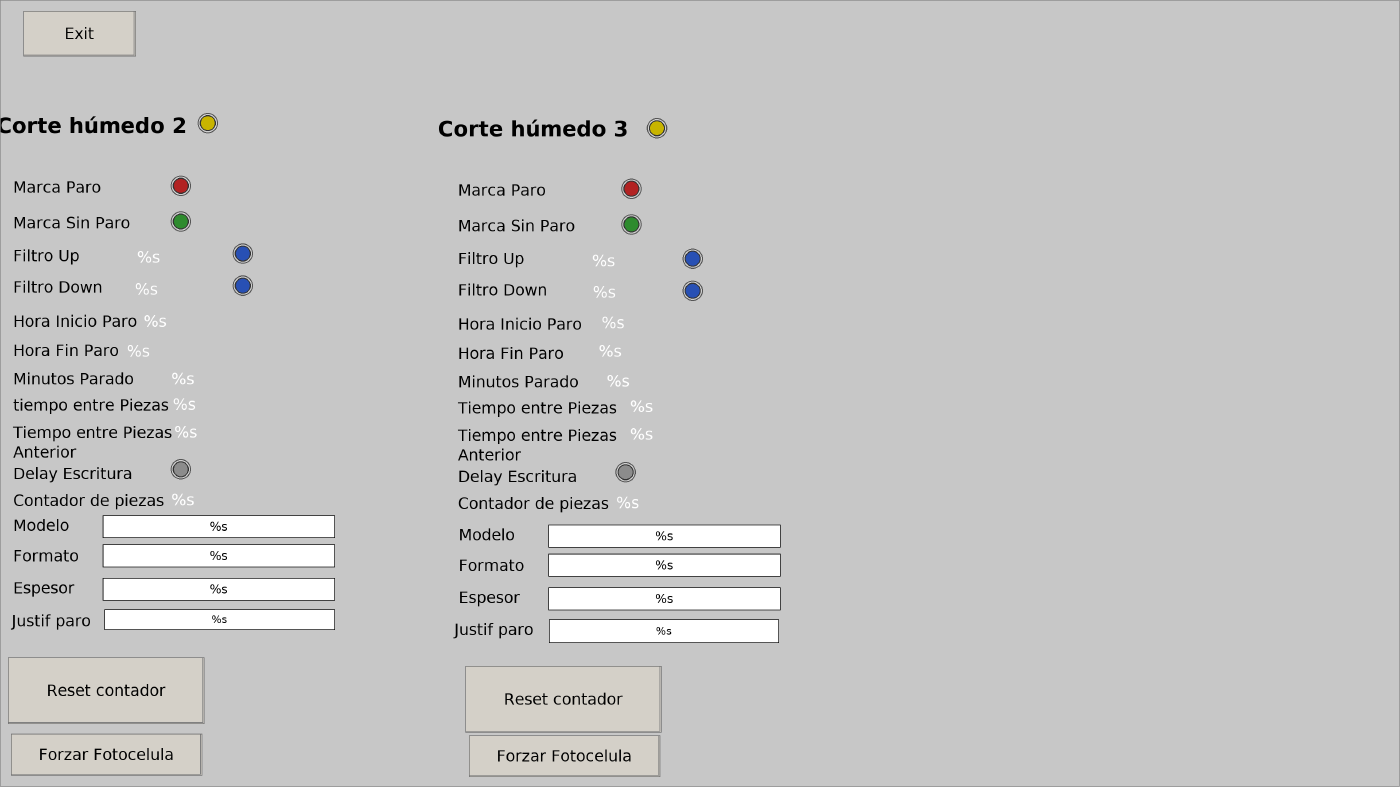
VISUALIZATION DiagnosticoFB  // 1920x1080
    Rectangle (185,338 93x30), "%s", text variable: FuncParoNodoRemote1CorteH2.Funci_CortHum2.tFiltro_up_Ftc.ET
    Label (10,146 231x53), "Corte húmedo 2"
    Label (15,242 150x30), "Marca Paro"
    Lamp1 (269,153 32x32), variable: FuncParoNodoRemote1CorteH2.Funci_CortHum2.Fotocelula, style: Lamp-Lamp1-Yellow
    Lamp1 (232,239 32x32), variable: FuncParoNodoRemote1CorteH2.Funci_CortHum2.MParo_Ftc, style: Lamp-Lamp1-Red
    Label (15,291 188x30), "Marca Sin Paro"
    Lamp1 (232,288 32x32), variable: FuncParoNodoRemote1CorteH2.Funci_CortHum2.M_SinParo_Ftc, style: Lamp-Lamp1-Green
    Label (15,336 117x30), "Filtro Up"
    Rectangle (182,382 93x30), "%s", text variable: FuncParoNodoRemote1CorteH2.Funci_CortHum2.tFiltro_down_Ftc.ET
    Label (15,379 143x30), "Filtro Down"
    Rectangle (194,426 183x30), "%s", text variable: FuncParoNodoRemote1CorteH2.Funci_CortHum2.H_InParo_Ftc
    Label (15,426 204x30), "Hora Inicio Paro"
    Lamp1 (317,332 32x32), variable: FuncParoNodoRemote1CorteH2.Funci_CortHum2.tFiltro_up_Ftc.Q, style: Lamp-Lamp1-Blue
    Lamp1 (317,376 32x32), variable: FuncParoNodoRemote1CorteH2.Funci_CortHum2.tFiltro_down_Ftc.Q, style: Lamp-Lamp1-Blue
    Rectangle (171,467 179x30), "%s", text variable: FuncParoNodoRemote1CorteH2.Funci_CortHum2.H_FinParo_Ftc
    Label (15,466 204x30), "Hora Fin Paro"
    Rectangle (232,505 192x30), "%s", text variable: FuncParoNodoRemote1CorteH2.Funci_CortHum2.Min_Parado_Ftc
    Label (15,505 204x30), "Minutos Parado"
    Label (15,541 244x30), "tiempo entre Piezas"
    Label (15,576 255x62), "Tiempo entre Piezas Anterior"
    Label (15,635 204x30), "Delay Escritura"
    Rectangle (232,671 93x30), "%s", text variable: FuncParoNodoRemote1CorteH2.Funci_CortHum2.Cont_Piezas_Ftc
    Label (15,672 215x30), "Contador de piezas"
    Lamp1 (232,628 32x32), variable: FuncParoNodoRemote1CorteH2.Funci_CortHum2.Delay_Esc_Ftc.Q, style: Lamp-Lamp1-Gray
    Button (32,15 154x62), "Exit"
        OnMouseClick: change screen: Home_CortH2
    Rectangle (809,343 93x30), "%s", text variable: FuncParoNodoLocalCorteH3.Funci_CortHum3.tFiltro_up_Ftc.ET
    Label (599,134 264x86), "Corte húmedo 3"
    Label (625,246 150x30), "Marca Paro"
    Lamp1 (885,160 32x32), variable: FuncParoNodoLocalCorteH3.Funci_CortHum3.Fotocelula, style: Lamp-Lamp1-Yellow
    Lamp1 (850,243 32x32), variable: FuncParoNodoLocalCorteH3.Funci_CortHum3.MParo_Ftc, style: Lamp-Lamp1-Red
    Label (625,295 188x30), "Marca Sin Paro"
    Lamp1 (850,292 32x32), variable: FuncParoNodoLocalCorteH3.Funci_CortHum3.M_SinParo_Ftc, style: Lamp-Lamp1-Green
    Label (625,340 117x30), "Filtro Up"
    Rectangle (810,386 93x30), "%s", text variable: FuncParoNodoLocalCorteH3.Funci_CortHum3.tFiltro_down_Ftc.ET
    Label (625,383 143x30), "Filtro Down"
    Rectangle (822,428 183x30), "%s", text variable: FuncParoNodoLocalCorteH3.Funci_CortHum3.H_InParo_Ftc
    Label (625,430 204x30), "Hora Inicio Paro"
    Lamp1 (934,339 32x32), variable: FuncParoNodoLocalCorteH3.Funci_CortHum3.tFiltro_up_Ftc.Q, style: Lamp-Lamp1-Blue
    Lamp1 (934,383 32x32), variable: FuncParoNodoLocalCorteH3.Funci_CortHum3.tFiltro_down_Ftc.Q, style: Lamp-Lamp1-Blue
    Rectangle (818,467 179x30), "%s", text variable: FuncParoNodoLocalCorteH3.Funci_CortHum3.H_FinParo_Ftc
    Label (625,470 204x30), "Hora Fin Paro"
    Rectangle (829,508 192x30), "%s", text variable: FuncParoNodoLocalCorteH3.Funci_CortHum3.Min_Parado_Ftc
    Label (625,509 204x30), "Minutos Parado"
    Label (625,545 244x30), "Tiempo entre Piezas"
    Label (625,580 255x62), "Tiempo entre Piezas Anterior"
    Label (625,639 204x30), "Delay Escritura"
    Rectangle (842,675 93x30), "%s", text variable: FuncParoNodoLocalCorteH3.Funci_CortHum3.Cont_Piezas_Ftc
    Label (625,676 215x30), "Contador de piezas"
    Lamp1 (842,632 32x32), variable: FuncParoNodoLocalCorteH3.Funci_CortHum3.Delay_Esc_Ftc.Q, style: Lamp-Lamp1-Gray
    Rectangle (234,540 192x30), "%s", text variable: FuncParoNodoRemote1CorteH2.Funci_CortHum2.t_Entre_Piez_Ftc
    Rectangle (861,543 192x30), "%s", text variable: FuncParoNodoLocalCorteH3.Funci_CortHum3.t_Entre_Piez_Ftc
    Rectangle (236,578 192x30), "%s", text variable: FuncParoNodoRemote1CorteH2.Funci_CortHum2.t_Entr_Piez_Ante_Ftc
    Rectangle (861,581 192x30), "%s", text variable: FuncParoNodoLocalCorteH3.Funci_CortHum3.t_Entr_Piez_Ante_Ftc
    Button (11,902 269x91), "Reset contador"
        tap FuncParoNodoRemote1CorteH2.Funci_CortHum2.ResetContPiez
    Button (638,914 269x91), "Reset contador"
        tap FuncParoNodoLocalCorteH3.Funci_CortHum3.ResetContPiez
    Button (643,1009 262x57), "Forzar Fotocelula"
        tap FuncParoNodoLocalCorteH3.ForzadoFtcCortHum3
    Button (15,1007 262x57), "Forzar Fotocelula"
        tap FuncParoNodoRemote1CorteH2.ForzadoFtcCortHum2
    Label (15,706 92x30), "Modelo"
    Label (15,748 105x30), "Formato"
    Label (15,792 99x30), "Espesor"
    Rectangle (141,707 318x31), "%s", text variable: FuncParoNodoRemote1CorteH2.FunGeneCortHum2.s_ModeloActualTabla
        OnMouseDown: write the text variable via Edit
    Rectangle (141,747 318x31), "%s", text variable: FuncParoNodoRemote1CorteH2.FunGeneCortHum2.s_FormatoActualTabla
        OnMouseDown: write the text variable via Edit
    Rectangle (141,793 318x31), "%s", text variable: FuncParoNodoRemote1CorteH2.FunGeneCortHum2.s_EspesorActualTabla
        OnMouseDown: write the text variable via Edit
    Label (626,719 92x30), "Modelo"
    Label (626,761 105x30), "Formato"
    Label (626,805 99x30), "Espesor"
    Rectangle (752,720 318x31), "%s", text variable: FuncParoNodoLocalCorteH3.FunGeneCortHum3.s_ModeloActualTabla
        OnMouseDown: write the text variable via Edit
    Rectangle (752,760 318x31), "%s", text variable: FuncParoNodoLocalCorteH3.FunGeneCortHum3.s_FormatoActualTabla
        OnMouseDown: write the text variable via Edit
    Rectangle (752,806 318x31), "%s", text variable: FuncParoNodoLocalCorteH3.FunGeneCortHum3.s_EspesorActualTabla
        OnMouseDown: write the text variable via Edit
    Label (13,837 123x30), "Justif paro"
    Rectangle (143,836 316x28), "%s", text variable: FuncParoNodoRemote1CorteH2.Funci_CortHum2.S_Justi_Paro_Ftc
        OnMouseDown: write the text variable via Edit
    Rectangle (753,850 315x32), "%s", text variable: FuncParoNodoLocalCorteH3.Funci_CortHum3.S_Justi_Paro_Ftc
        OnMouseDown: write the text variable via Edit
    Label (620,849 123x30), "Justif paro"
END_VISUALIZATION

(* stored: Version 1.1.0.1, ProductVersion 3.1.4024.12
   Visu DiagnosticoFB: Id {0e784541-fdbe-4048-8d88-3d9ad672f9bb} *)
